# EPICS autosave request: urRobotApp/Db/path_settings.req
$(P)PathPvFile.VAL
$(P)PathPvDescFile.VAL
